// TIA Portal V19 export
VAR_GLOBAL   // PLC tag table "Loop1_IO"
   Loop1_LsConnectorPlugged AT %I130.5 : Bool;   // 920S1
   Loop1_LsMaxLow AT %I130.7 : Bool;   // 920S2
   Loop1_LsMinHigh AT %I130.6 : Bool;   // 920S1
   Ansa1_Coprifossa_V_Salita AT %Q132.3 : Bool;   // 922YV1
   Ansa1_Coprifossa_V_Discesa AT %Q132.4 : Bool;   // 922YV2
   Ansa1_Coprifossa_Ls_Alto AT %I131.0 : Bool;   // 922SQ1
   Ansa1_Coprifossa_Ls_Basso AT %I131.1 : Bool;   // 922SQ2
   Ansa1_Coprifossa_Ls_Libero AT %I131.2 : Bool;   // 922
END_VAR
